(* PLC project SafeLOGIC-1, BrAutomation SafeDESIGNER  4.3.2.11 *)
(* stored: companyURL http://www.br-automation.com, creationDateTime Mon Apr 30 13:16:50 2018 *)

PROGRAM Main
  VAR  (* added by the conversion: wires and edge detectors of the diagram *)
    _AND_S23_OUT : ANY;
  END_VAR

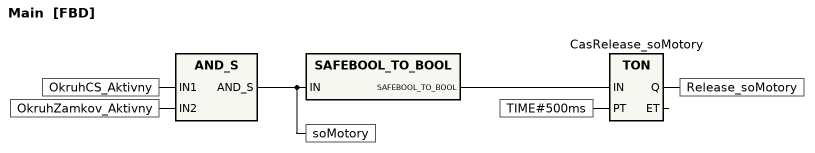
(* FBD diagram, written out as Structured Text *)
_AND_S23_OUT := AND_S(OkruhCS_Aktivny, OkruhZamkov_Aktivny);
soMotory := _AND_S23_OUT;
CasRelease_soMotory(IN := SAFEBOOL_TO_BOOL(_AND_S23_OUT), PT := TIME#500ms);
Release_soMotory := CasRelease_soMotory.Q;
END_PROGRAM
